// TIA Portal V17 export
// export: Created 2026-04-13T11:12:53.4230829Z, ExportSetting WithDefaults, DisplayName Totally Integrated Automation Portal, DisplayVersion V17 Update 4, DisplayName TIA Portal Openness, DisplayVersion V17 Update 4, DisplayName TIA Portal Version Control Interface, DisplayVersion V17, DisplayName SINAMICS Startdrive Advanced, DisplayVersion V17, DisplayName SINAMICS Startdrive G130, G150, S120, S150, SINAMICS MV, S210, DisplayVersion V17, DisplayName SINAMICS Startdrive G110M, G120, G120C, G120D, G120P, G115D, DisplayVersion V17, DisplayName STEP 7 Professional, DisplayVersion V17 Update 4, DisplayName STEP 7 Safety, DisplayVersion V17, DisplayName WinCC Professional, DisplayVersion V17 Update 4
TagTable "INCIPJS"
  INCIPJS_1设定时间 : Real  (PLC tag INCIPJS.1设定时间, HMI_连接_1, 1 s)
  INCIPJS_2设定时间 : Real  (PLC tag INCIPJS.2设定时间, HMI_连接_1, 1 s)
  INCIPJS_3设定时间 : Real  (PLC tag INCIPJS.3设定时间, HMI_连接_1, 1 s)
  INCIPJS_4设定时间 : Real  (PLC tag INCIPJS.4设定时间, HMI_连接_1, 1 s)
  INCIPJS_5设定时间 : Real  (PLC tag INCIPJS.5设定时间, HMI_连接_1, 1 s)
  INCIPJS_6设定时间 : Real  (PLC tag INCIPJS.6设定时间, HMI_连接_1, 1 s)
  INCIPJS_7设定时间 : Real  (PLC tag INCIPJS.7设定时间, HMI_连接_1, 1 s)
  INCIPJS_8设定时间 : Real  (PLC tag INCIPJS.8设定时间, HMI_连接_1, 1 s)
  INCIPJS_9设定时间 : Real  (PLC tag INCIPJS.9设定时间, HMI_连接_1, 1 s)
  INCIPJS_10设定时间 : Real  (PLC tag INCIPJS.10设定时间, HMI_连接_1, 1 s)
  INCIPJS_11设定时间 : Real  (PLC tag INCIPJS.11设定时间, HMI_连接_1, 1 s)
  INCIPJS_12设定时间 : Real  (PLC tag INCIPJS.12设定时间, HMI_连接_1, 1 s)
  INCIPJS_13设定时间 : Real  (PLC tag INCIPJS.13设定时间, HMI_连接_1, 1 s)
  INCIPJS_14设定时间 : Real  (PLC tag INCIPJS.14设定时间, HMI_连接_1, 1 s)
  INCIPJS_15设定时间 : Real  (PLC tag INCIPJS.15设定时间, HMI_连接_1, 1 s)
  INCIPJS_16设定时间 : Real  (PLC tag INCIPJS.16设定时间, HMI_连接_1, 1 s)
  INCIPJS_1计时 : Real  (PLC tag INCIPJS.1计时, HMI_连接_1, 1 s)
  INCIPJS_2计时 : Real  (PLC tag INCIPJS.2计时, HMI_连接_1, 1 s)
  INCIPJS_3计时 : Real  (PLC tag INCIPJS.3计时, HMI_连接_1, 1 s)
  INCIPJS_4计时 : Real  (PLC tag INCIPJS.4计时, HMI_连接_1, 1 s)
  INCIPJS_5计时 : Real  (PLC tag INCIPJS.5计时, HMI_连接_1, 1 s)
  INCIPJS_6计时 : Real  (PLC tag INCIPJS.6计时, HMI_连接_1, 1 s)
  INCIPJS_7计时 : Real  (PLC tag INCIPJS.7计时, HMI_连接_1, 1 s)
  INCIPJS_8计时 : Real  (PLC tag INCIPJS.8计时, HMI_连接_1, 1 s)
  INCIPJS_9计时 : Real  (PLC tag INCIPJS.9计时, HMI_连接_1, 1 s)
  INCIPJS_10计时 : Real  (PLC tag INCIPJS.10计时, HMI_连接_1, 1 s)
  INCIPJS_11计时 : Real  (PLC tag INCIPJS.11计时, HMI_连接_1, 1 s)
  INCIPJS_12计时 : Real  (PLC tag INCIPJS.12计时, HMI_连接_1, 1 s)
  INCIPJS_13计时 : Real  (PLC tag INCIPJS.13计时, HMI_连接_1, 1 s)
  INCIPJS_14计时 : Real  (PLC tag INCIPJS.14计时, HMI_连接_1, 1 s)
  INCIPJS_15计时 : Real  (PLC tag INCIPJS.15计时, HMI_连接_1, 1 s)
  INCIPJS_16计时 : Real  (PLC tag INCIPJS.16计时, HMI_连接_1, 1 s)
